// TIA Portal project "FactoryIO_Template_S7-1500_V15_parcial1_terminado1" (V15)

(* hardware
DEVICE "S71500/ET200MP-Station_1"  S7-1500 station
   slot 0: "Profilschiene_0"  6ES7 590-1***0-0AA0
   slot 1: "PLC_1"  CPU 1511-1 PN  6ES7 511-1AK00-0AB0  V1.8
   slot 2: "AI 8xU/I/RTD/TC ST_1"  AI 8xU/I/RTD/TC ST  6ES7 531-7KF00-0AB0  V2.0
   slot 3: "AI 8xU/I/RTD/TC ST_2"  AI 8xU/I/RTD/TC ST  6ES7 531-7KF00-0AB0  V2.0
   slot 4: "AI 8xU/I/RTD/TC ST_3"  AI 8xU/I/RTD/TC ST  6ES7 531-7KF00-0AB0  V2.0
   slot 5: "AI 8xU/I/RTD/TC ST_4"  AI 8xU/I/RTD/TC ST  6ES7 531-7KF00-0AB0  V2.0
   slot 6: "DI 16x24VDC BA_1"  DI 16x24VDC BA  6ES7 521-1BH10-0AA0  V1.0
*)

// ===== PLC "PLC_1"  CPU 1511-1 PN =====

VAR_GLOBAL   // PLC tag table "Standard-Variablentabelle"
   "Box_feeder" AT %Q0.0 : Bool;
   "Load_belt" AT %Q0.1 : Bool;
   "Start" AT %I0.0 : Bool;
   "Stop" AT %I0.1 : Bool;
   "Reset" AT %I0.2 : Bool;
   "Manual" AT %I0.3 : Bool;
   "Emergency_stop" AT %I0.5 : Bool;
   "Box_entry" AT %I0.6 : Bool;
   "Turn" AT %Q0.2 : Bool;
   "Pusher_limit" AT %I0.7 : Bool;
   "Push" AT %Q0.3 : Bool;
   "Open_Plate" AT %Q0.4 : Bool;
   "Plate_limit" AT %I1.0 : Bool;
   "Clamp" AT %Q0.5 : Bool;
   "Clamped" AT %I1.1 : Bool;
   "Pallet_feeder" AT %Q0.6 : Bool;
   "Pallet_at_entry" AT %I1.2 : Bool;
   "S1_Elevator_base" AT %I1.3 : Bool;
   "S2_Elevator_base" AT %I1.4 : Bool;
   "Pallet_at_exit" AT %I1.5 : Bool;
   "Exit_conveyor" AT %Q0.7 : Bool;
   "Elevator_moving" AT %I1.6 : Bool;
   "Move_to_limit" AT %Q1.0 : Bool;
   "Elevator_up" AT %Q1.1 : Bool;
   "Warning light" AT %Q1.3 : Bool;
   "Auto" AT %I0.4 : Bool;
   "Elevator_down" AT %Q1.2 : Bool;
   "Contador1" AT %MW10 : Int;
   "Contador2" AT %MW12 : Int;
   "Contador3" AT %MW14 : Int;
   "LimiteContador1" AT %MW20 : Int;
   "LimiteContador2" AT %MW22 : Int;
   "Pallet_in_acensor" AT %M100.0 : Bool;
   "Load_pallet" AT %Q1.4 : Bool;
   "Run_machine" AT %M0.0 : Bool;
   "Elevator_Listo_a_cargar" AT %M100.1 : Bool;
   "LimiteContador3" AT %MW24 : Int;
   "Plaforma_llena" AT %M100.2 : Bool;
   "Reposo" AT %M1000.0 : Bool;
   "Bandas_on" AT %M1000.1 : Bool;
   "Caja_en_posicion" AT %M1000.2 : Bool;
   "box_hacia_load_belt" AT %M1000.3 : Bool;
   "Avanzando_en_box_en_load_belt" AT %M1000.4 : Bool;
   "Haciendo_push" AT %M1000.5 : Bool;
   "Saliendo_push" AT %M1000.6 : Bool;
   "Push_afuera" AT %M1000.7 : Bool;
   "Push_regresando" AT %M1001.0 : Bool;
   "Push_en_inicio" AT %M1001.1 : Bool;
   "Cajas_en_plato" AT %M1001.2 : Bool;
   "Intercambiar_con_turn" AT %M1001.3 : Bool;
   "Intercambiar_sin_turn" AT %M1001.4 : Bool;
   "Reposo_inferiror" AT %M1100.0 : Bool;
   "Pallet_avanzando" AT %M1100.1 : Bool;
   "Entrando_a_load_pallet" AT %M1100.2 : Bool;
   "Pallet_en_posicion" AT %M1100.3 : Bool;
   "Acomodar_pallet" AT %M1100.4 : Bool;
   "Pallet_in_acesor_op" AT %M1100.5 : Bool;
   "Muevo_ascensor" AT %M1100.6 : Bool;
   "acesor_subiendo" AT %M1100.7 : Bool;
   "elevator_arriba" AT %M1101.0 : Bool;
   "Empezar_descarga_activar_clamp" AT %M1101.1 : Bool;
   "cajas_sujetas_a_descargar" AT %M1101.2 : Bool;
   "plate_abriendo" AT %M1101.3 : Bool;
   "plate_abierto" AT %M1101.4 : Bool;
   "Cajas_en_pallet" AT %M1101.5 : Bool;
   "elevator_bajando" AT %M1101.6 : Bool;
   "elevator_bajo_1" AT %M1101.7 : Bool;
   "Cerrando_plato" AT %M1102.0 : Bool;
   "plato_cerrado" AT %M1102.1 : Bool;
   "Elevador_lleno" AT %M1102.2 : Bool;
   "Acensor_bajando" AT %M1102.3 : Bool;
   "Asensor_abajo" AT %M1102.4 : Bool;
   "Pallet_Saliendo_de_elevador" AT %M1102.5 : Bool;
   "Restableciendo_inicio" AT %M1102.6 : Bool;
   "EstadosRdePCajas1" AT %MB1000 : Byte;
   "EstadosRdePEstibas1" AT %MB1100 : Byte;
   "EstadosRdePCajas2" AT %MB1001 : Byte;
   "MemEstadosRdePCajas1" AT %MB2000 : Byte;
   "MemEstadosRdePCajas2" AT %MB2001 : Byte;
   "MemEstadosRdePEstibas1" AT %MB2100 : Byte;
   "EstadosRdePEstibas2" AT %MB1101 : Byte;
   "EstadosRdePEstibas3" AT %MB1102 : Byte;
   "MemEstadosRdePEstibas2" AT %MB2101 : Byte;
   "MemEstadosRdePEstibas3" AT %MB2102 : Byte;
   "Salidas_Byte_0" AT %QB0 : Byte;
   "MemSalidas_Byte_0" AT %MB3000 : Byte;
   "Salidas_Byte_1" AT %QB1 : Byte;
   "MemSalidas_Byte_1" AT %MB3001 : Byte;
   "Tag_1" AT %M900.0 : Bool;
   "Tag_3" AT %M900.1 : Bool;
   "EstadosMaquina1" AT %MB100 : Byte;
   "MemEstadosMaquina1" AT %MB4000 : Byte;
   "Estado_On_Machine" AT %MB0 : Byte;
   "MenEstado_On_Machine" AT %MB5000 : Byte;
   "Entrada_POT" AT %ID30 : Real;
   "Salida_contador" AT %QD30 : Real;
   "Pot_int" AT %MW2 : Int;
   "Pallet_Feeder_Aux" AT %Q1.5 : Bool;
   "Roller_Stop" AT %Q1.6 : Bool;
END_VAR

// folder: System blocks/Program resources

DATA_BLOCK "Contador_1"   // DB1
{ S7_Optimized_Access := 'TRUE' }
AUTHOR : Simatic
FAMILY : IEC
NAME : CNTR
VERSION : 1.0
// stored: InstanceOfName IEC_COUNTER
"IEC_COUNTER"
BEGIN
END_DATA_BLOCK

DATA_BLOCK "Contador_2"   // DB2
{ S7_Optimized_Access := 'TRUE' }
AUTHOR : Simatic
FAMILY : IEC
NAME : CNTR
VERSION : 1.0
// stored: InstanceOfName IEC_COUNTER
"IEC_COUNTER"
BEGIN
END_DATA_BLOCK

DATA_BLOCK "Contador_3"   // DB3
{ S7_Optimized_Access := 'TRUE' }
AUTHOR : Simatic
FAMILY : IEC
NAME : CNTR
VERSION : 1.0
// stored: InstanceOfName IEC_COUNTER
"IEC_COUNTER"
BEGIN
END_DATA_BLOCK

// folder: (top level)

FUNCTION "Nivel_superior" : Void   // FC1, LAD
{ S7_Optimized_Access := 'TRUE' }
VERSION : 0.1
   VAR_TEMP   // added for the SCL form of the ladder/FBD networks
      _w1 : Bool;
   END_VAR
BEGIN

REGION Network 1
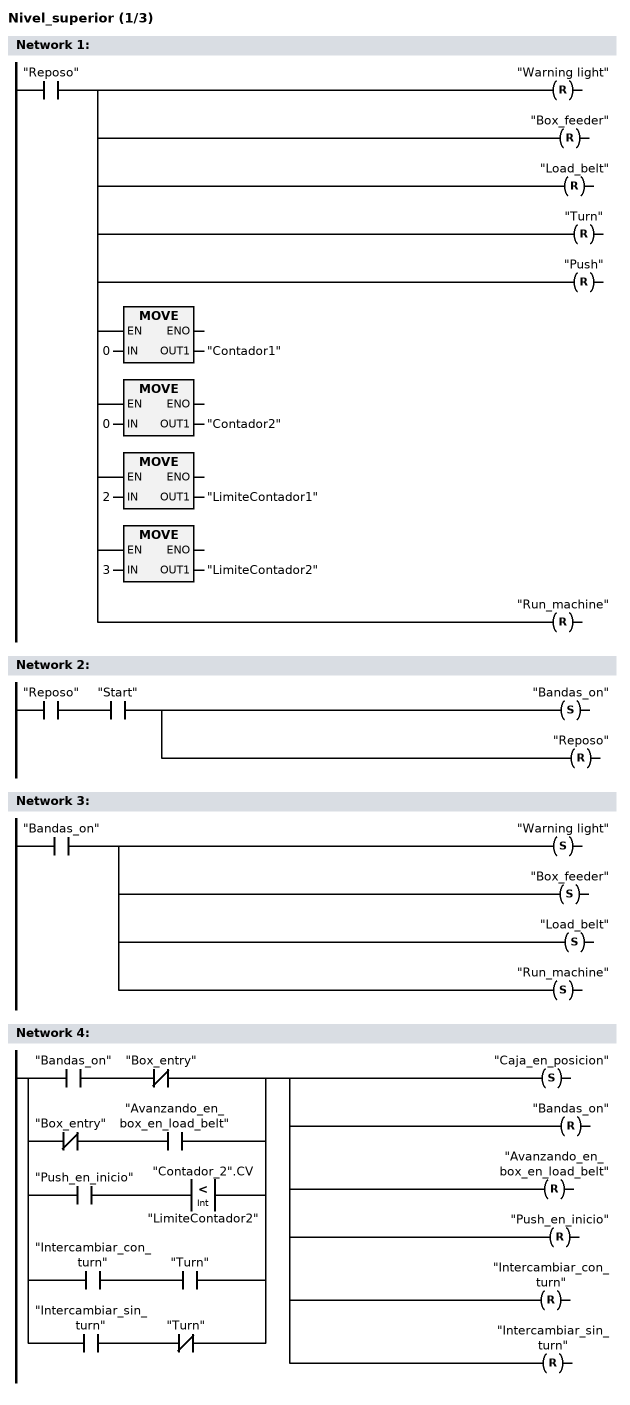
   RUNG wire#powerrail
      Contact( "Reposo" )
      wire#w1
      R_Coil( "Warning light" )
   END_RUNG
   RUNG wire#w1
      R_Coil( "Box_feeder" )
   END_RUNG
   RUNG wire#w1
      R_Coil( "Load_belt" )
   END_RUNG
   RUNG wire#w1
      R_Coil( "Turn" )
   END_RUNG
   RUNG wire#w1
      R_Coil( "Push" )
   END_RUNG
   RUNG wire#w1
      Move(in := 0, out1 => "Contador1")
   END_RUNG
   RUNG wire#w1
      Move(in := 0, out1 => "Contador2")
   END_RUNG
   RUNG wire#w1
      Move(in := 2, out1 => "LimiteContador1")
   END_RUNG
   RUNG wire#w1
      Move(in := 3, out1 => "LimiteContador2")
   END_RUNG
   RUNG wire#w1
      R_Coil( "Run_machine" )
   END_RUNG
   // the same network as SCL:
   IF "Reposo" THEN
       "Warning light" := FALSE;
       "Box_feeder" := FALSE;
       "Load_belt" := FALSE;
       "Turn" := FALSE;
       "Push" := FALSE;
       "Contador1" := 0;
       "Contador2" := 0;
       "LimiteContador1" := 2;
       "LimiteContador2" := 3;
       "Run_machine" := FALSE;
   END_IF;
END_REGION

REGION Network 2
   RUNG wire#powerrail
      Contact( "Reposo" )
      Contact( "Start" )
      wire#w1
      S_Coil( "Bandas_on" )
   END_RUNG
   RUNG wire#w1
      R_Coil( "Reposo" )
   END_RUNG
   // the same network as SCL:
   IF "Reposo" AND "Start" THEN
       "Bandas_on" := TRUE;
       "Reposo" := FALSE;
   END_IF;
END_REGION

REGION Network 3
   RUNG wire#powerrail
      Contact( "Bandas_on" )
      wire#w1
      S_Coil( "Warning light" )
   END_RUNG
   RUNG wire#w1
      S_Coil( "Box_feeder" )
   END_RUNG
   RUNG wire#w1
      S_Coil( "Load_belt" )
   END_RUNG
   RUNG wire#w1
      S_Coil( "Run_machine" )
   END_RUNG
   // the same network as SCL:
   IF "Bandas_on" THEN
       "Warning light" := TRUE;
       "Box_feeder" := TRUE;
       "Load_belt" := TRUE;
       "Run_machine" := TRUE;
   END_IF;
END_REGION

REGION Network 4
   RUNG wire#powerrail
      Contact( "Bandas_on" )
      I_Contact( "Box_entry" )
      wire#w1
      S_Coil( "Caja_en_posicion" )
   END_RUNG
   RUNG wire#powerrail
      I_Contact( "Box_entry" )
      Contact( "Avanzando_en_box_en_load_belt" )
   END_RUNG wire#w1
   RUNG wire#powerrail
      Contact( "Push_en_inicio" )
      { S7_Templates := "SrcType := Int" } LT_Contact(in1 := "Contador_2".CV, in2 := "LimiteContador2")
   END_RUNG wire#w1
   RUNG wire#powerrail
      Contact( "Intercambiar_con_turn" )
      Contact( "Turn" )
   END_RUNG wire#w1
   RUNG wire#powerrail
      Contact( "Intercambiar_sin_turn" )
      I_Contact( "Turn" )
   END_RUNG wire#w1
   RUNG wire#w1
      R_Coil( "Bandas_on" )
   END_RUNG
   RUNG wire#w1
      R_Coil( "Avanzando_en_box_en_load_belt" )
   END_RUNG
   RUNG wire#w1
      R_Coil( "Push_en_inicio" )
   END_RUNG
   RUNG wire#w1
      R_Coil( "Intercambiar_con_turn" )
   END_RUNG
   RUNG wire#w1
      R_Coil( "Intercambiar_sin_turn" )
   END_RUNG
   // the same network as SCL:
   IF ("Bandas_on" AND NOT "Box_entry") OR (NOT "Box_entry" AND "Avanzando_en_box_en_load_belt") OR ("Push_en_inicio" AND ("Contador_2".CV < "LimiteContador2")) OR ("Intercambiar_con_turn" AND "Turn") OR ("Intercambiar_sin_turn" AND NOT "Turn") THEN
       "Caja_en_posicion" := TRUE;
   END_IF;
   #_w1 := ("Bandas_on" AND NOT "Box_entry") OR (NOT "Box_entry" AND "Avanzando_en_box_en_load_belt") OR ("Push_en_inicio" AND ("Contador_2".CV < "LimiteContador2")) OR ("Intercambiar_con_turn" AND "Turn") OR ("Intercambiar_sin_turn" AND NOT "Turn");
   IF #_w1 THEN
       "Bandas_on" := FALSE;
       "Avanzando_en_box_en_load_belt" := FALSE;
       "Push_en_inicio" := FALSE;
       "Intercambiar_con_turn" := FALSE;
       "Intercambiar_sin_turn" := FALSE;
   END_IF;
END_REGION

REGION Network 5
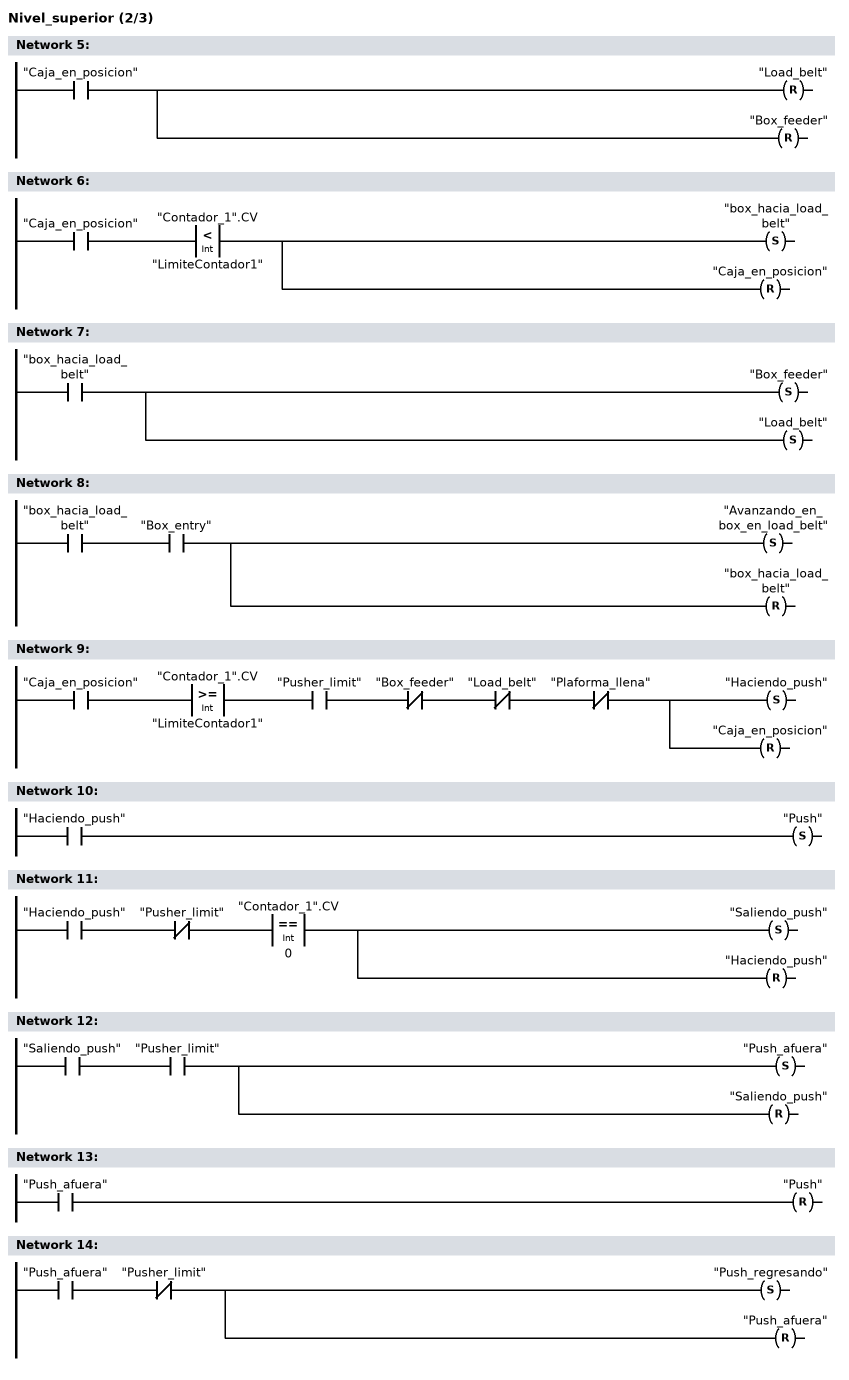
   RUNG wire#powerrail
      Contact( "Caja_en_posicion" )
      wire#w1
      R_Coil( "Load_belt" )
   END_RUNG
   RUNG wire#w1
      R_Coil( "Box_feeder" )
   END_RUNG
   // the same network as SCL:
   IF "Caja_en_posicion" THEN
       "Load_belt" := FALSE;
       "Box_feeder" := FALSE;
   END_IF;
END_REGION

REGION Network 6
   RUNG wire#powerrail
      Contact( "Caja_en_posicion" )
      { S7_Templates := "SrcType := Int" } LT_Contact(in1 := "Contador_1".CV, in2 := "LimiteContador1")
      wire#w1
      S_Coil( "box_hacia_load_belt" )
   END_RUNG
   RUNG wire#w1
      R_Coil( "Caja_en_posicion" )
   END_RUNG
   // the same network as SCL:
   IF "Caja_en_posicion" AND ("Contador_1".CV < "LimiteContador1") THEN
       "box_hacia_load_belt" := TRUE;
       "Caja_en_posicion" := FALSE;
   END_IF;
END_REGION

REGION Network 7
   RUNG wire#powerrail
      Contact( "box_hacia_load_belt" )
      wire#w1
      S_Coil( "Box_feeder" )
   END_RUNG
   RUNG wire#w1
      S_Coil( "Load_belt" )
   END_RUNG
   // the same network as SCL:
   IF "box_hacia_load_belt" THEN
       "Box_feeder" := TRUE;
       "Load_belt" := TRUE;
   END_IF;
END_REGION

REGION Network 8
   RUNG wire#powerrail
      Contact( "box_hacia_load_belt" )
      Contact( "Box_entry" )
      wire#w1
      S_Coil( "Avanzando_en_box_en_load_belt" )
   END_RUNG
   RUNG wire#w1
      R_Coil( "box_hacia_load_belt" )
   END_RUNG
   // the same network as SCL:
   IF "box_hacia_load_belt" AND "Box_entry" THEN
       "Avanzando_en_box_en_load_belt" := TRUE;
       "box_hacia_load_belt" := FALSE;
   END_IF;
END_REGION

REGION Network 9
   RUNG wire#powerrail
      Contact( "Caja_en_posicion" )
      { S7_Templates := "SrcType := Int" } GE_Contact(in1 := "Contador_1".CV, in2 := "LimiteContador1")
      Contact( "Pusher_limit" )
      I_Contact( "Box_feeder" )
      I_Contact( "Load_belt" )
      I_Contact( "Plaforma_llena" )
      wire#w1
      S_Coil( "Haciendo_push" )
   END_RUNG
   RUNG wire#w1
      R_Coil( "Caja_en_posicion" )
   END_RUNG
   // the same network as SCL:
   IF "Caja_en_posicion" AND ("Contador_1".CV >= "LimiteContador1") AND "Pusher_limit" AND NOT "Box_feeder" AND NOT "Load_belt" AND NOT "Plaforma_llena" THEN
       "Haciendo_push" := TRUE;
       "Caja_en_posicion" := FALSE;
   END_IF;
END_REGION

REGION Network 10
   RUNG wire#powerrail
      Contact( "Haciendo_push" )
      S_Coil( "Push" )
   END_RUNG
   // the same network as SCL:
   IF "Haciendo_push" THEN "Push" := TRUE; END_IF;
END_REGION

REGION Network 11
   RUNG wire#powerrail
      Contact( "Haciendo_push" )
      I_Contact( "Pusher_limit" )
      { S7_Templates := "SrcType := Int" } EQ_Contact(in1 := "Contador_1".CV, in2 := 0)
      wire#w1
      S_Coil( "Saliendo_push" )
   END_RUNG
   RUNG wire#w1
      R_Coil( "Haciendo_push" )
   END_RUNG
   // the same network as SCL:
   IF "Haciendo_push" AND NOT "Pusher_limit" AND ("Contador_1".CV = 0) THEN
       "Saliendo_push" := TRUE;
       "Haciendo_push" := FALSE;
   END_IF;
END_REGION

REGION Network 12
   RUNG wire#powerrail
      Contact( "Saliendo_push" )
      Contact( "Pusher_limit" )
      wire#w1
      S_Coil( "Push_afuera" )
   END_RUNG
   RUNG wire#w1
      R_Coil( "Saliendo_push" )
   END_RUNG
   // the same network as SCL:
   IF "Saliendo_push" AND "Pusher_limit" THEN
       "Push_afuera" := TRUE;
       "Saliendo_push" := FALSE;
   END_IF;
END_REGION

REGION Network 13
   RUNG wire#powerrail
      Contact( "Push_afuera" )
      R_Coil( "Push" )
   END_RUNG
   // the same network as SCL:
   IF "Push_afuera" THEN "Push" := FALSE; END_IF;
END_REGION

REGION Network 14
   RUNG wire#powerrail
      Contact( "Push_afuera" )
      I_Contact( "Pusher_limit" )
      wire#w1
      S_Coil( "Push_regresando" )
   END_RUNG
   RUNG wire#w1
      R_Coil( "Push_afuera" )
   END_RUNG
   // the same network as SCL:
   IF "Push_afuera" AND NOT "Pusher_limit" THEN
       "Push_regresando" := TRUE;
       "Push_afuera" := FALSE;
   END_IF;
END_REGION

REGION Network 15
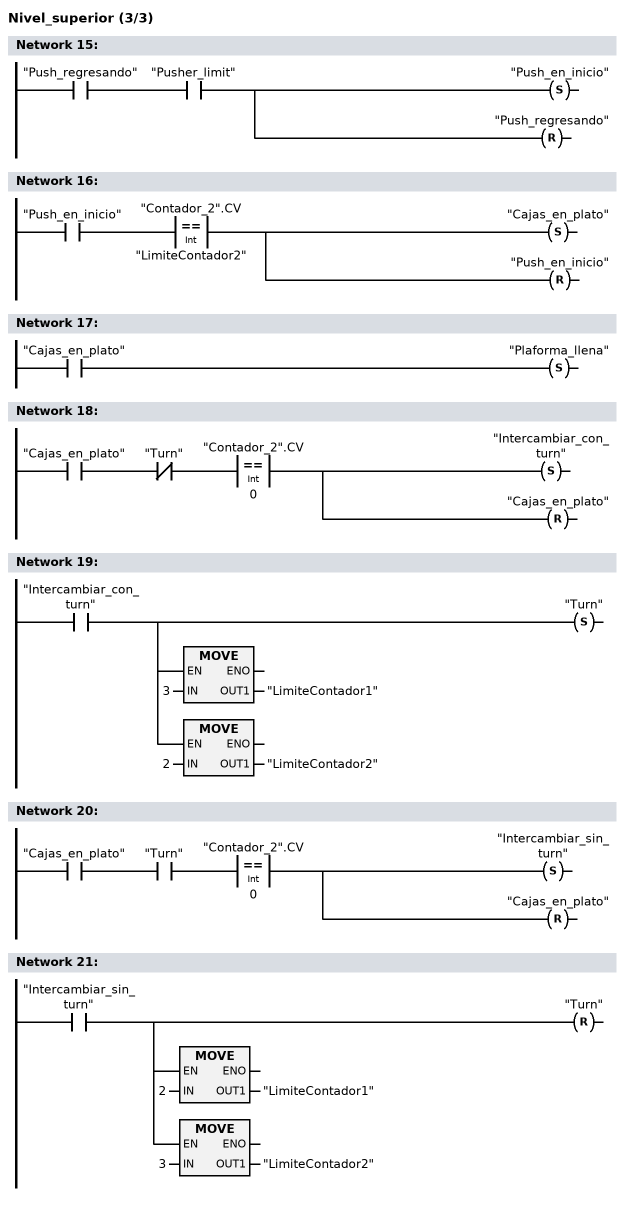
   RUNG wire#powerrail
      Contact( "Push_regresando" )
      Contact( "Pusher_limit" )
      wire#w1
      S_Coil( "Push_en_inicio" )
   END_RUNG
   RUNG wire#w1
      R_Coil( "Push_regresando" )
   END_RUNG
   // the same network as SCL:
   IF "Push_regresando" AND "Pusher_limit" THEN
       "Push_en_inicio" := TRUE;
       "Push_regresando" := FALSE;
   END_IF;
END_REGION

REGION Network 16
   RUNG wire#powerrail
      Contact( "Push_en_inicio" )
      { S7_Templates := "SrcType := Int" } EQ_Contact(in1 := "Contador_2".CV, in2 := "LimiteContador2")
      wire#w1
      S_Coil( "Cajas_en_plato" )
   END_RUNG
   RUNG wire#w1
      R_Coil( "Push_en_inicio" )
   END_RUNG
   // the same network as SCL:
   IF "Push_en_inicio" AND ("Contador_2".CV = "LimiteContador2") THEN
       "Cajas_en_plato" := TRUE;
       "Push_en_inicio" := FALSE;
   END_IF;
END_REGION

REGION Network 17
   RUNG wire#powerrail
      Contact( "Cajas_en_plato" )
      S_Coil( "Plaforma_llena" )
   END_RUNG
   // the same network as SCL:
   IF "Cajas_en_plato" THEN "Plaforma_llena" := TRUE; END_IF;
END_REGION

REGION Network 18
   RUNG wire#powerrail
      Contact( "Cajas_en_plato" )
      I_Contact( "Turn" )
      { S7_Templates := "SrcType := Int" } EQ_Contact(in1 := "Contador_2".CV, in2 := 0)
      wire#w1
      S_Coil( "Intercambiar_con_turn" )
   END_RUNG
   RUNG wire#w1
      R_Coil( "Cajas_en_plato" )
   END_RUNG
   // the same network as SCL:
   IF "Cajas_en_plato" AND NOT "Turn" AND ("Contador_2".CV = 0) THEN
       "Intercambiar_con_turn" := TRUE;
       "Cajas_en_plato" := FALSE;
   END_IF;
END_REGION

REGION Network 19
   RUNG wire#powerrail
      Contact( "Intercambiar_con_turn" )
      wire#w1
      S_Coil( "Turn" )
   END_RUNG
   RUNG wire#w1
      Move(in := 3, out1 => "LimiteContador1")
   END_RUNG
   RUNG wire#w1
      Move(in := 2, out1 => "LimiteContador2")
   END_RUNG
   // the same network as SCL:
   IF "Intercambiar_con_turn" THEN
       "Turn" := TRUE;
       "LimiteContador1" := 3;
       "LimiteContador2" := 2;
   END_IF;
END_REGION

REGION Network 20
   RUNG wire#powerrail
      Contact( "Cajas_en_plato" )
      Contact( "Turn" )
      { S7_Templates := "SrcType := Int" } EQ_Contact(in1 := "Contador_2".CV, in2 := 0)
      wire#w1
      S_Coil( "Intercambiar_sin_turn" )
   END_RUNG
   RUNG wire#w1
      R_Coil( "Cajas_en_plato" )
   END_RUNG
   // the same network as SCL:
   IF "Cajas_en_plato" AND "Turn" AND ("Contador_2".CV = 0) THEN
       "Intercambiar_sin_turn" := TRUE;
       "Cajas_en_plato" := FALSE;
   END_IF;
END_REGION

REGION Network 21
   RUNG wire#powerrail
      Contact( "Intercambiar_sin_turn" )
      wire#w1
      R_Coil( "Turn" )
   END_RUNG
   RUNG wire#w1
      Move(in := 2, out1 => "LimiteContador1")
   END_RUNG
   RUNG wire#w1
      Move(in := 3, out1 => "LimiteContador2")
   END_RUNG
   // the same network as SCL:
   IF "Intercambiar_sin_turn" THEN
       "Turn" := FALSE;
       "LimiteContador1" := 2;
       "LimiteContador2" := 3;
   END_IF;
END_REGION
END_FUNCTION

FUNCTION "Nivel_inferior" : Void   // FC2, LAD
{ S7_Optimized_Access := 'TRUE' }
VERSION : 0.1
   VAR_TEMP   // added for the SCL form of the ladder/FBD networks
      _w1 : Bool;
   END_VAR
BEGIN

REGION Network 1
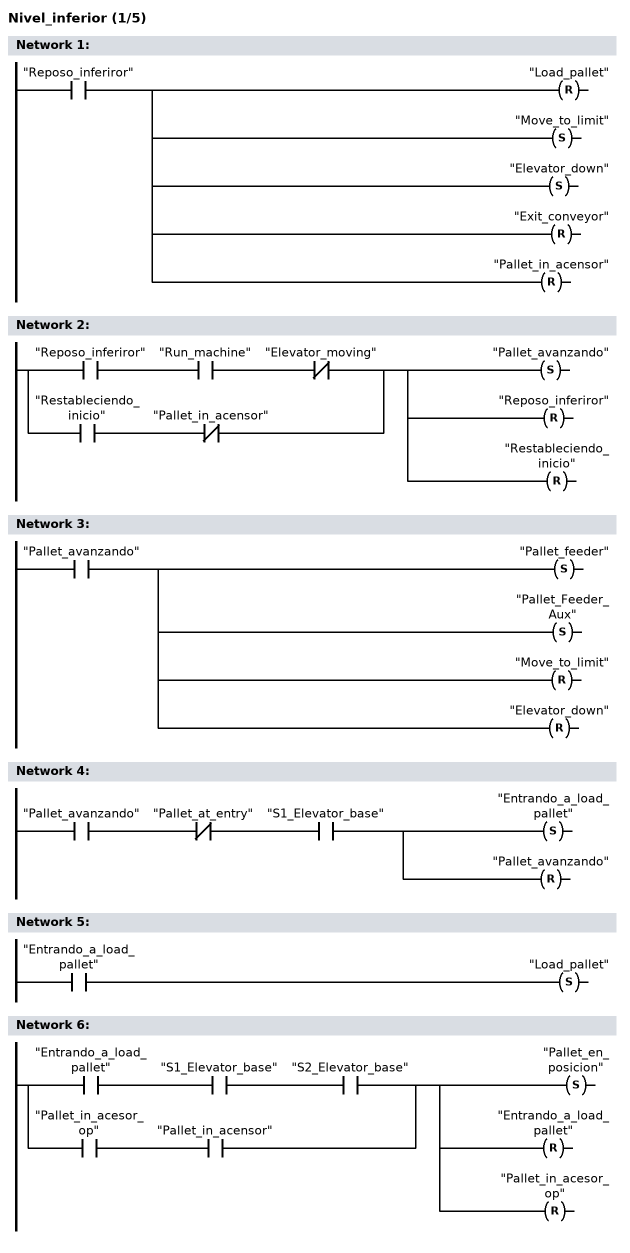
   RUNG wire#powerrail
      Contact( "Reposo_inferiror" )
      wire#w1
      R_Coil( "Load_pallet" )
   END_RUNG
   RUNG wire#w1
      S_Coil( "Move_to_limit" )
   END_RUNG
   RUNG wire#w1
      S_Coil( "Elevator_down" )
   END_RUNG
   RUNG wire#w1
      R_Coil( "Exit_conveyor" )
   END_RUNG
   RUNG wire#w1
      R_Coil( "Pallet_in_acensor" )
   END_RUNG
   // the same network as SCL:
   IF "Reposo_inferiror" THEN
       "Load_pallet" := FALSE;
       "Move_to_limit" := TRUE;
       "Elevator_down" := TRUE;
       "Exit_conveyor" := FALSE;
       "Pallet_in_acensor" := FALSE;
   END_IF;
END_REGION

REGION Network 2
   RUNG wire#powerrail
      Contact( "Reposo_inferiror" )
      Contact( "Run_machine" )
      I_Contact( "Elevator_moving" )
      wire#w1
      S_Coil( "Pallet_avanzando" )
   END_RUNG
   RUNG wire#powerrail
      Contact( "Restableciendo_inicio" )
      I_Contact( "Pallet_in_acensor" )
   END_RUNG wire#w1
   RUNG wire#w1
      R_Coil( "Reposo_inferiror" )
   END_RUNG
   RUNG wire#w1
      R_Coil( "Restableciendo_inicio" )
   END_RUNG
   // the same network as SCL:
   IF ("Reposo_inferiror" AND "Run_machine" AND NOT "Elevator_moving") OR ("Restableciendo_inicio" AND NOT "Pallet_in_acensor") THEN
       "Pallet_avanzando" := TRUE;
   END_IF;
   #_w1 := ("Reposo_inferiror" AND "Run_machine" AND NOT "Elevator_moving") OR ("Restableciendo_inicio" AND NOT "Pallet_in_acensor");
   IF #_w1 THEN
       "Reposo_inferiror" := FALSE;
       "Restableciendo_inicio" := FALSE;
   END_IF;
END_REGION

REGION Network 3
   RUNG wire#powerrail
      Contact( "Pallet_avanzando" )
      wire#w1
      S_Coil( "Pallet_feeder" )
   END_RUNG
   RUNG wire#w1
      S_Coil( "Pallet_Feeder_Aux" )
   END_RUNG
   RUNG wire#w1
      R_Coil( "Move_to_limit" )
   END_RUNG
   RUNG wire#w1
      R_Coil( "Elevator_down" )
   END_RUNG
   // the same network as SCL:
   IF "Pallet_avanzando" THEN
       "Pallet_feeder" := TRUE;
       "Pallet_Feeder_Aux" := TRUE;
       "Move_to_limit" := FALSE;
       "Elevator_down" := FALSE;
   END_IF;
END_REGION

REGION Network 4
   RUNG wire#powerrail
      Contact( "Pallet_avanzando" )
      I_Contact( "Pallet_at_entry" )
      Contact( "S1_Elevator_base" )
      wire#w1
      S_Coil( "Entrando_a_load_pallet" )
   END_RUNG
   RUNG wire#w1
      R_Coil( "Pallet_avanzando" )
   END_RUNG
   // the same network as SCL:
   IF "Pallet_avanzando" AND NOT "Pallet_at_entry" AND "S1_Elevator_base" THEN
       "Entrando_a_load_pallet" := TRUE;
       "Pallet_avanzando" := FALSE;
   END_IF;
END_REGION

REGION Network 5
   RUNG wire#powerrail
      Contact( "Entrando_a_load_pallet" )
      S_Coil( "Load_pallet" )
   END_RUNG
   // the same network as SCL:
   IF "Entrando_a_load_pallet" THEN "Load_pallet" := TRUE; END_IF;
END_REGION

REGION Network 6
   RUNG wire#powerrail
      Contact( "Entrando_a_load_pallet" )
      Contact( "S1_Elevator_base" )
      Contact( "S2_Elevator_base" )
      wire#w1
      S_Coil( "Pallet_en_posicion" )
   END_RUNG
   RUNG wire#powerrail
      Contact( "Pallet_in_acesor_op" )
      Contact( "Pallet_in_acensor" )
   END_RUNG wire#w1
   RUNG wire#w1
      R_Coil( "Entrando_a_load_pallet" )
   END_RUNG
   RUNG wire#w1
      R_Coil( "Pallet_in_acesor_op" )
   END_RUNG
   // the same network as SCL:
   IF ("Entrando_a_load_pallet" AND "S1_Elevator_base" AND "S2_Elevator_base") OR ("Pallet_in_acesor_op" AND "Pallet_in_acensor") THEN
       "Pallet_en_posicion" := TRUE;
   END_IF;
   #_w1 := ("Entrando_a_load_pallet" AND "S1_Elevator_base" AND "S2_Elevator_base") OR ("Pallet_in_acesor_op" AND "Pallet_in_acensor");
   IF #_w1 THEN
       "Entrando_a_load_pallet" := FALSE;
       "Pallet_in_acesor_op" := FALSE;
   END_IF;
END_REGION

REGION Network 7
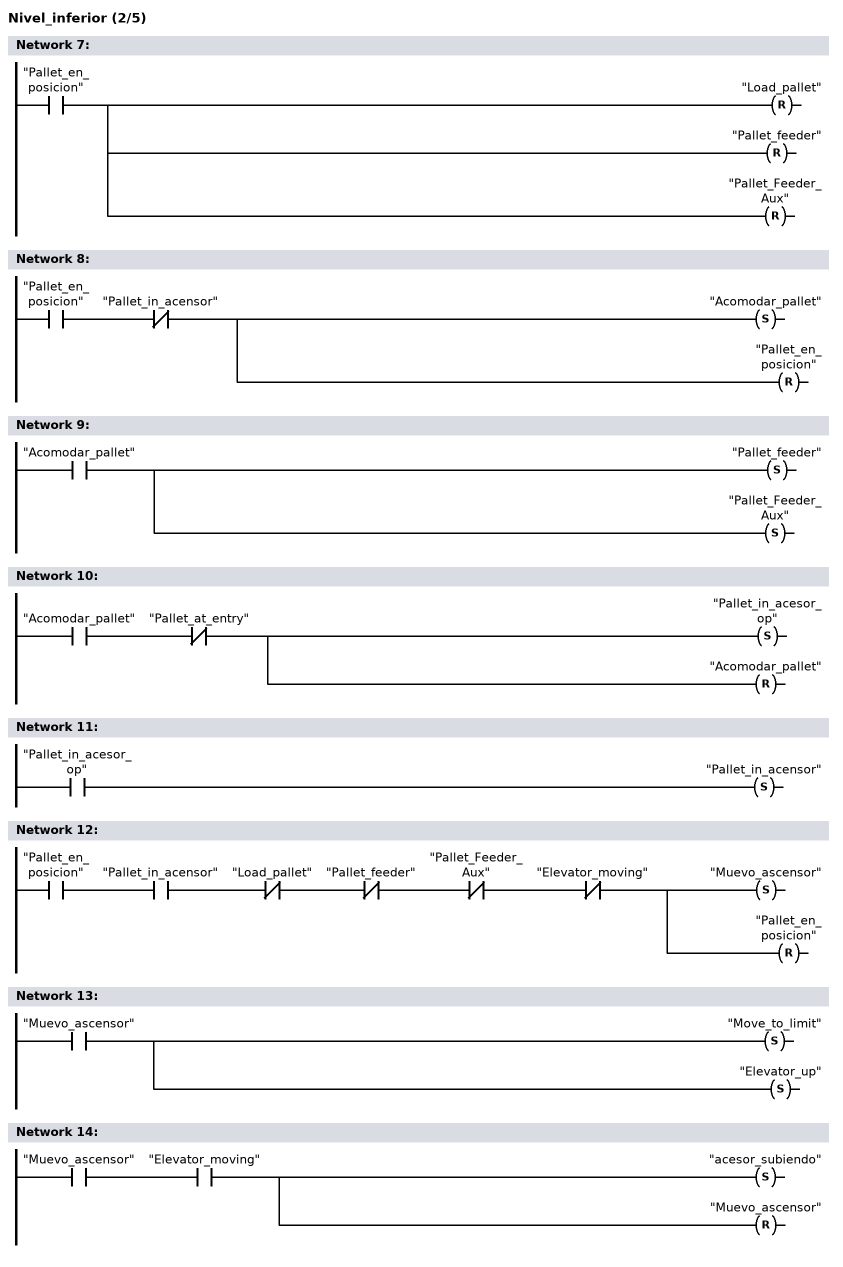
   RUNG wire#powerrail
      Contact( "Pallet_en_posicion" )
      wire#w1
      R_Coil( "Load_pallet" )
   END_RUNG
   RUNG wire#w1
      R_Coil( "Pallet_feeder" )
   END_RUNG
   RUNG wire#w1
      R_Coil( "Pallet_Feeder_Aux" )
   END_RUNG
   // the same network as SCL:
   IF "Pallet_en_posicion" THEN
       "Load_pallet" := FALSE;
       "Pallet_feeder" := FALSE;
       "Pallet_Feeder_Aux" := FALSE;
   END_IF;
END_REGION

REGION Network 8
   RUNG wire#powerrail
      Contact( "Pallet_en_posicion" )
      I_Contact( "Pallet_in_acensor" )
      wire#w1
      S_Coil( "Acomodar_pallet" )
   END_RUNG
   RUNG wire#w1
      R_Coil( "Pallet_en_posicion" )
   END_RUNG
   // the same network as SCL:
   IF "Pallet_en_posicion" AND NOT "Pallet_in_acensor" THEN
       "Acomodar_pallet" := TRUE;
       "Pallet_en_posicion" := FALSE;
   END_IF;
END_REGION

REGION Network 9
   RUNG wire#powerrail
      Contact( "Acomodar_pallet" )
      wire#w1
      S_Coil( "Pallet_feeder" )
   END_RUNG
   RUNG wire#w1
      S_Coil( "Pallet_Feeder_Aux" )
   END_RUNG
   // the same network as SCL:
   IF "Acomodar_pallet" THEN
       "Pallet_feeder" := TRUE;
       "Pallet_Feeder_Aux" := TRUE;
   END_IF;
END_REGION

REGION Network 10
   RUNG wire#powerrail
      Contact( "Acomodar_pallet" )
      I_Contact( "Pallet_at_entry" )
      wire#w1
      S_Coil( "Pallet_in_acesor_op" )
   END_RUNG
   RUNG wire#w1
      R_Coil( "Acomodar_pallet" )
   END_RUNG
   // the same network as SCL:
   IF "Acomodar_pallet" AND NOT "Pallet_at_entry" THEN
       "Pallet_in_acesor_op" := TRUE;
       "Acomodar_pallet" := FALSE;
   END_IF;
END_REGION

REGION Network 11
   RUNG wire#powerrail
      Contact( "Pallet_in_acesor_op" )
      S_Coil( "Pallet_in_acensor" )
   END_RUNG
   // the same network as SCL:
   IF "Pallet_in_acesor_op" THEN "Pallet_in_acensor" := TRUE; END_IF;
END_REGION

REGION Network 12
   RUNG wire#powerrail
      Contact( "Pallet_en_posicion" )
      Contact( "Pallet_in_acensor" )
      I_Contact( "Load_pallet" )
      I_Contact( "Pallet_feeder" )
      I_Contact( "Pallet_Feeder_Aux" )
      I_Contact( "Elevator_moving" )
      wire#w1
      S_Coil( "Muevo_ascensor" )
   END_RUNG
   RUNG wire#w1
      R_Coil( "Pallet_en_posicion" )
   END_RUNG
   // the same network as SCL:
   IF "Pallet_en_posicion" AND "Pallet_in_acensor" AND NOT "Load_pallet" AND NOT "Pallet_feeder" AND NOT "Pallet_Feeder_Aux" AND NOT "Elevator_moving" THEN
       "Muevo_ascensor" := TRUE;
       "Pallet_en_posicion" := FALSE;
   END_IF;
END_REGION

REGION Network 13
   RUNG wire#powerrail
      Contact( "Muevo_ascensor" )
      wire#w1
      S_Coil( "Move_to_limit" )
   END_RUNG
   RUNG wire#w1
      S_Coil( "Elevator_up" )
   END_RUNG
   // the same network as SCL:
   IF "Muevo_ascensor" THEN
       "Move_to_limit" := TRUE;
       "Elevator_up" := TRUE;
   END_IF;
END_REGION

REGION Network 14
   RUNG wire#powerrail
      Contact( "Muevo_ascensor" )
      Contact( "Elevator_moving" )
      wire#w1
      S_Coil( "acesor_subiendo" )
   END_RUNG
   RUNG wire#w1
      R_Coil( "Muevo_ascensor" )
   END_RUNG
   // the same network as SCL:
   IF "Muevo_ascensor" AND "Elevator_moving" THEN
       "acesor_subiendo" := TRUE;
       "Muevo_ascensor" := FALSE;
   END_IF;
END_REGION

REGION Network 15
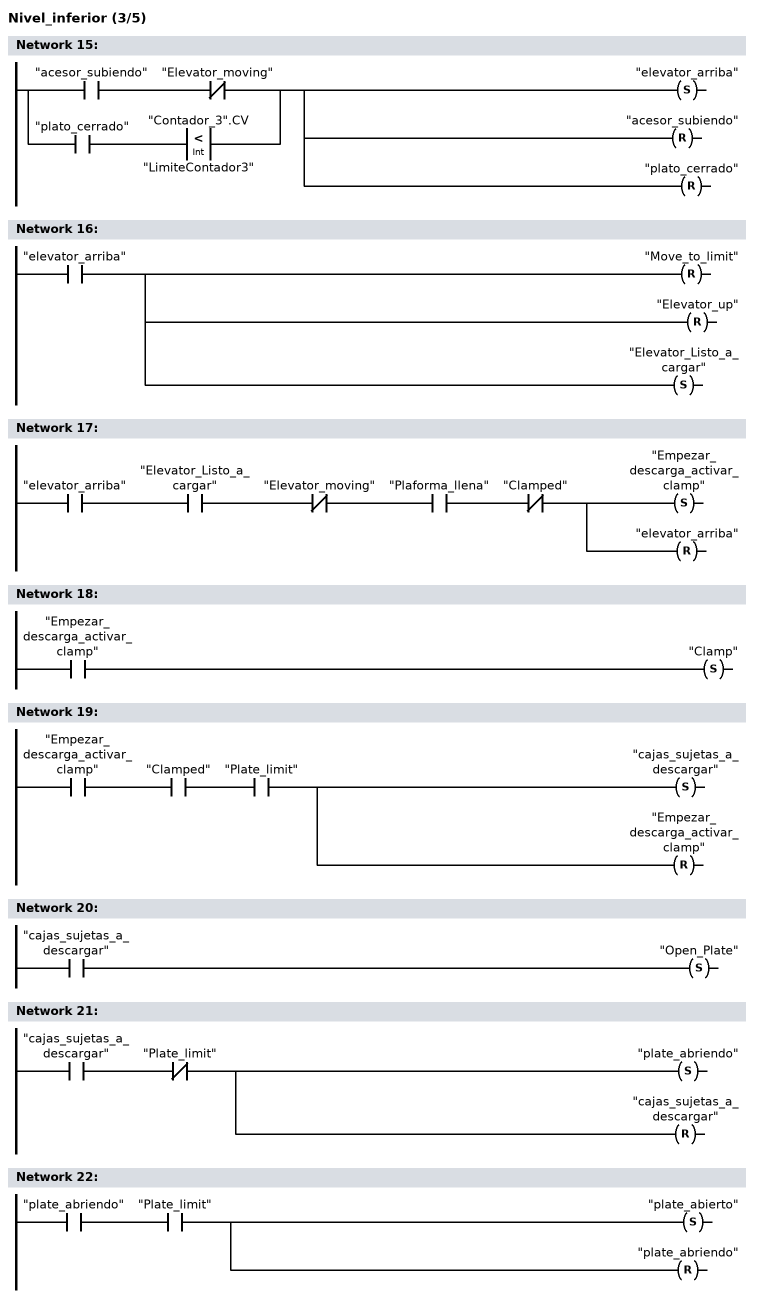
   RUNG wire#powerrail
      Contact( "acesor_subiendo" )
      I_Contact( "Elevator_moving" )
      wire#w1
      S_Coil( "elevator_arriba" )
   END_RUNG
   RUNG wire#powerrail
      Contact( "plato_cerrado" )
      { S7_Templates := "SrcType := Int" } LT_Contact(in1 := "Contador_3".CV, in2 := "LimiteContador3")
   END_RUNG wire#w1
   RUNG wire#w1
      R_Coil( "acesor_subiendo" )
   END_RUNG
   RUNG wire#w1
      R_Coil( "plato_cerrado" )
   END_RUNG
   // the same network as SCL:
   IF ("acesor_subiendo" AND NOT "Elevator_moving") OR ("plato_cerrado" AND ("Contador_3".CV < "LimiteContador3")) THEN
       "elevator_arriba" := TRUE;
   END_IF;
   #_w1 := ("acesor_subiendo" AND NOT "Elevator_moving") OR ("plato_cerrado" AND ("Contador_3".CV < "LimiteContador3"));
   IF #_w1 THEN
       "acesor_subiendo" := FALSE;
       "plato_cerrado" := FALSE;
   END_IF;
END_REGION

REGION Network 16
   RUNG wire#powerrail
      Contact( "elevator_arriba" )
      wire#w1
      R_Coil( "Move_to_limit" )
   END_RUNG
   RUNG wire#w1
      R_Coil( "Elevator_up" )
   END_RUNG
   RUNG wire#w1
      S_Coil( "Elevator_Listo_a_cargar" )
   END_RUNG
   // the same network as SCL:
   IF "elevator_arriba" THEN
       "Move_to_limit" := FALSE;
       "Elevator_up" := FALSE;
       "Elevator_Listo_a_cargar" := TRUE;
   END_IF;
END_REGION

REGION Network 17
   RUNG wire#powerrail
      Contact( "elevator_arriba" )
      Contact( "Elevator_Listo_a_cargar" )
      I_Contact( "Elevator_moving" )
      Contact( "Plaforma_llena" )
      I_Contact( "Clamped" )
      wire#w1
      S_Coil( "Empezar_descarga_activar_clamp" )
   END_RUNG
   RUNG wire#w1
      R_Coil( "elevator_arriba" )
   END_RUNG
   // the same network as SCL:
   IF "elevator_arriba" AND "Elevator_Listo_a_cargar" AND NOT "Elevator_moving" AND "Plaforma_llena" AND NOT "Clamped" THEN
       "Empezar_descarga_activar_clamp" := TRUE;
       "elevator_arriba" := FALSE;
   END_IF;
END_REGION

REGION Network 18
   RUNG wire#powerrail
      Contact( "Empezar_descarga_activar_clamp" )
      S_Coil( "Clamp" )
   END_RUNG
   // the same network as SCL:
   IF "Empezar_descarga_activar_clamp" THEN "Clamp" := TRUE; END_IF;
END_REGION

REGION Network 19
   RUNG wire#powerrail
      Contact( "Empezar_descarga_activar_clamp" )
      Contact( "Clamped" )
      Contact( "Plate_limit" )
      wire#w1
      S_Coil( "cajas_sujetas_a_descargar" )
   END_RUNG
   RUNG wire#w1
      R_Coil( "Empezar_descarga_activar_clamp" )
   END_RUNG
   // the same network as SCL:
   IF "Empezar_descarga_activar_clamp" AND "Clamped" AND "Plate_limit" THEN
       "cajas_sujetas_a_descargar" := TRUE;
       "Empezar_descarga_activar_clamp" := FALSE;
   END_IF;
END_REGION

REGION Network 20
   RUNG wire#powerrail
      Contact( "cajas_sujetas_a_descargar" )
      S_Coil( "Open_Plate" )
   END_RUNG
   // the same network as SCL:
   IF "cajas_sujetas_a_descargar" THEN "Open_Plate" := TRUE; END_IF;
END_REGION

REGION Network 21
   RUNG wire#powerrail
      Contact( "cajas_sujetas_a_descargar" )
      I_Contact( "Plate_limit" )
      wire#w1
      S_Coil( "plate_abriendo" )
   END_RUNG
   RUNG wire#w1
      R_Coil( "cajas_sujetas_a_descargar" )
   END_RUNG
   // the same network as SCL:
   IF "cajas_sujetas_a_descargar" AND NOT "Plate_limit" THEN
       "plate_abriendo" := TRUE;
       "cajas_sujetas_a_descargar" := FALSE;
   END_IF;
END_REGION

REGION Network 22
   RUNG wire#powerrail
      Contact( "plate_abriendo" )
      Contact( "Plate_limit" )
      wire#w1
      S_Coil( "plate_abierto" )
   END_RUNG
   RUNG wire#w1
      R_Coil( "plate_abriendo" )
   END_RUNG
   // the same network as SCL:
   IF "plate_abriendo" AND "Plate_limit" THEN
       "plate_abierto" := TRUE;
       "plate_abriendo" := FALSE;
   END_IF;
END_REGION

REGION Network 23
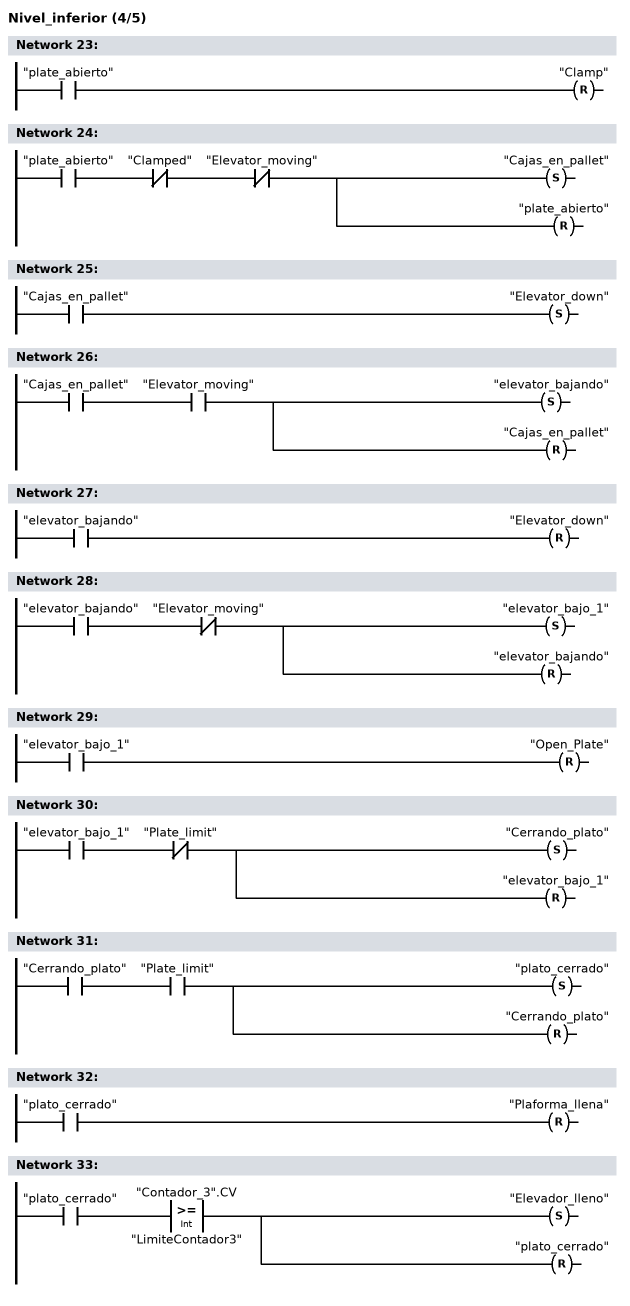
   RUNG wire#powerrail
      Contact( "plate_abierto" )
      R_Coil( "Clamp" )
   END_RUNG
   // the same network as SCL:
   IF "plate_abierto" THEN "Clamp" := FALSE; END_IF;
END_REGION

REGION Network 24
   RUNG wire#powerrail
      Contact( "plate_abierto" )
      I_Contact( "Clamped" )
      I_Contact( "Elevator_moving" )
      wire#w1
      S_Coil( "Cajas_en_pallet" )
   END_RUNG
   RUNG wire#w1
      R_Coil( "plate_abierto" )
   END_RUNG
   // the same network as SCL:
   IF "plate_abierto" AND NOT "Clamped" AND NOT "Elevator_moving" THEN
       "Cajas_en_pallet" := TRUE;
       "plate_abierto" := FALSE;
   END_IF;
END_REGION

REGION Network 25
   RUNG wire#powerrail
      Contact( "Cajas_en_pallet" )
      S_Coil( "Elevator_down" )
   END_RUNG
   // the same network as SCL:
   IF "Cajas_en_pallet" THEN "Elevator_down" := TRUE; END_IF;
END_REGION

REGION Network 26
   RUNG wire#powerrail
      Contact( "Cajas_en_pallet" )
      Contact( "Elevator_moving" )
      wire#w1
      S_Coil( "elevator_bajando" )
   END_RUNG
   RUNG wire#w1
      R_Coil( "Cajas_en_pallet" )
   END_RUNG
   // the same network as SCL:
   IF "Cajas_en_pallet" AND "Elevator_moving" THEN
       "elevator_bajando" := TRUE;
       "Cajas_en_pallet" := FALSE;
   END_IF;
END_REGION

REGION Network 27
   RUNG wire#powerrail
      Contact( "elevator_bajando" )
      R_Coil( "Elevator_down" )
   END_RUNG
   // the same network as SCL:
   IF "elevator_bajando" THEN "Elevator_down" := FALSE; END_IF;
END_REGION

REGION Network 28
   RUNG wire#powerrail
      Contact( "elevator_bajando" )
      I_Contact( "Elevator_moving" )
      wire#w1
      S_Coil( "elevator_bajo_1" )
   END_RUNG
   RUNG wire#w1
      R_Coil( "elevator_bajando" )
   END_RUNG
   // the same network as SCL:
   IF "elevator_bajando" AND NOT "Elevator_moving" THEN
       "elevator_bajo_1" := TRUE;
       "elevator_bajando" := FALSE;
   END_IF;
END_REGION

REGION Network 29
   RUNG wire#powerrail
      Contact( "elevator_bajo_1" )
      R_Coil( "Open_Plate" )
   END_RUNG
   // the same network as SCL:
   IF "elevator_bajo_1" THEN "Open_Plate" := FALSE; END_IF;
END_REGION

REGION Network 30
   RUNG wire#powerrail
      Contact( "elevator_bajo_1" )
      I_Contact( "Plate_limit" )
      wire#w1
      S_Coil( "Cerrando_plato" )
   END_RUNG
   RUNG wire#w1
      R_Coil( "elevator_bajo_1" )
   END_RUNG
   // the same network as SCL:
   IF "elevator_bajo_1" AND NOT "Plate_limit" THEN
       "Cerrando_plato" := TRUE;
       "elevator_bajo_1" := FALSE;
   END_IF;
END_REGION

REGION Network 31
   RUNG wire#powerrail
      Contact( "Cerrando_plato" )
      Contact( "Plate_limit" )
      wire#w1
      S_Coil( "plato_cerrado" )
   END_RUNG
   RUNG wire#w1
      R_Coil( "Cerrando_plato" )
   END_RUNG
   // the same network as SCL:
   IF "Cerrando_plato" AND "Plate_limit" THEN
       "plato_cerrado" := TRUE;
       "Cerrando_plato" := FALSE;
   END_IF;
END_REGION

REGION Network 32
   RUNG wire#powerrail
      Contact( "plato_cerrado" )
      R_Coil( "Plaforma_llena" )
   END_RUNG
   // the same network as SCL:
   IF "plato_cerrado" THEN "Plaforma_llena" := FALSE; END_IF;
END_REGION

REGION Network 33
   RUNG wire#powerrail
      Contact( "plato_cerrado" )
      { S7_Templates := "SrcType := Int" } GE_Contact(in1 := "Contador_3".CV, in2 := "LimiteContador3")
      wire#w1
      S_Coil( "Elevador_lleno" )
   END_RUNG
   RUNG wire#w1
      R_Coil( "plato_cerrado" )
   END_RUNG
   // the same network as SCL:
   IF "plato_cerrado" AND ("Contador_3".CV >= "LimiteContador3") THEN
       "Elevador_lleno" := TRUE;
       "plato_cerrado" := FALSE;
   END_IF;
END_REGION

REGION Network 34
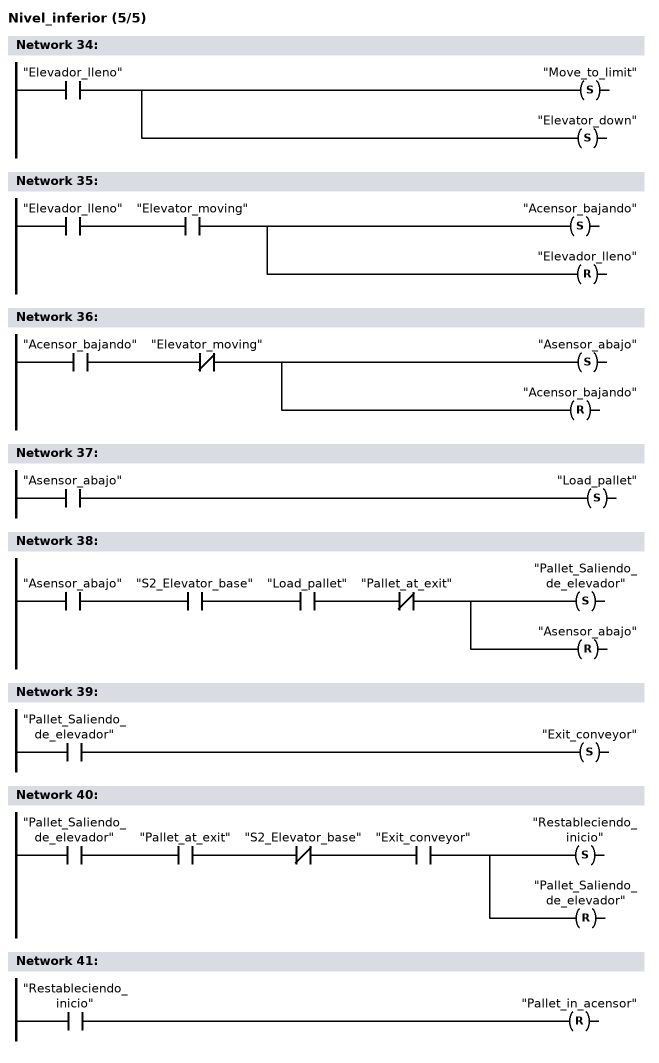
   RUNG wire#powerrail
      Contact( "Elevador_lleno" )
      wire#w1
      S_Coil( "Move_to_limit" )
   END_RUNG
   RUNG wire#w1
      S_Coil( "Elevator_down" )
   END_RUNG
   // the same network as SCL:
   IF "Elevador_lleno" THEN
       "Move_to_limit" := TRUE;
       "Elevator_down" := TRUE;
   END_IF;
END_REGION

REGION Network 35
   RUNG wire#powerrail
      Contact( "Elevador_lleno" )
      Contact( "Elevator_moving" )
      wire#w1
      S_Coil( "Acensor_bajando" )
   END_RUNG
   RUNG wire#w1
      R_Coil( "Elevador_lleno" )
   END_RUNG
   // the same network as SCL:
   IF "Elevador_lleno" AND "Elevator_moving" THEN
       "Acensor_bajando" := TRUE;
       "Elevador_lleno" := FALSE;
   END_IF;
END_REGION

REGION Network 36
   RUNG wire#powerrail
      Contact( "Acensor_bajando" )
      I_Contact( "Elevator_moving" )
      wire#w1
      S_Coil( "Asensor_abajo" )
   END_RUNG
   RUNG wire#w1
      R_Coil( "Acensor_bajando" )
   END_RUNG
   // the same network as SCL:
   IF "Acensor_bajando" AND NOT "Elevator_moving" THEN
       "Asensor_abajo" := TRUE;
       "Acensor_bajando" := FALSE;
   END_IF;
END_REGION

REGION Network 37
   RUNG wire#powerrail
      Contact( "Asensor_abajo" )
      S_Coil( "Load_pallet" )
   END_RUNG
   // the same network as SCL:
   IF "Asensor_abajo" THEN "Load_pallet" := TRUE; END_IF;
END_REGION

REGION Network 38
   RUNG wire#powerrail
      Contact( "Asensor_abajo" )
      Contact( "S2_Elevator_base" )
      Contact( "Load_pallet" )
      I_Contact( "Pallet_at_exit" )
      wire#w1
      S_Coil( "Pallet_Saliendo_de_elevador" )
   END_RUNG
   RUNG wire#w1
      R_Coil( "Asensor_abajo" )
   END_RUNG
   // the same network as SCL:
   IF "Asensor_abajo" AND "S2_Elevator_base" AND "Load_pallet" AND NOT "Pallet_at_exit" THEN
       "Pallet_Saliendo_de_elevador" := TRUE;
       "Asensor_abajo" := FALSE;
   END_IF;
END_REGION

REGION Network 39
   RUNG wire#powerrail
      Contact( "Pallet_Saliendo_de_elevador" )
      S_Coil( "Exit_conveyor" )
   END_RUNG
   // the same network as SCL:
   IF "Pallet_Saliendo_de_elevador" THEN "Exit_conveyor" := TRUE; END_IF;
END_REGION

REGION Network 40
   RUNG wire#powerrail
      Contact( "Pallet_Saliendo_de_elevador" )
      Contact( "Pallet_at_exit" )
      I_Contact( "S2_Elevator_base" )
      Contact( "Exit_conveyor" )
      wire#w1
      S_Coil( "Restableciendo_inicio" )
   END_RUNG
   RUNG wire#w1
      R_Coil( "Pallet_Saliendo_de_elevador" )
   END_RUNG
   // the same network as SCL:
   IF "Pallet_Saliendo_de_elevador" AND "Pallet_at_exit" AND NOT "S2_Elevator_base" AND "Exit_conveyor" THEN
       "Restableciendo_inicio" := TRUE;
       "Pallet_Saliendo_de_elevador" := FALSE;
   END_IF;
END_REGION

REGION Network 41
   RUNG wire#powerrail
      Contact( "Restableciendo_inicio" )
      R_Coil( "Pallet_in_acensor" )
   END_RUNG
   // the same network as SCL:
   IF "Restableciendo_inicio" THEN "Pallet_in_acensor" := FALSE; END_IF;
END_REGION
END_FUNCTION

FUNCTION "Contadores" : Void   // FC3, LAD
{ S7_Optimized_Access := 'TRUE' }
VERSION : 0.1
   VAR_TEMP
      TEMP_salida_conta : Real;
   END_VAR
BEGIN

REGION Network 1
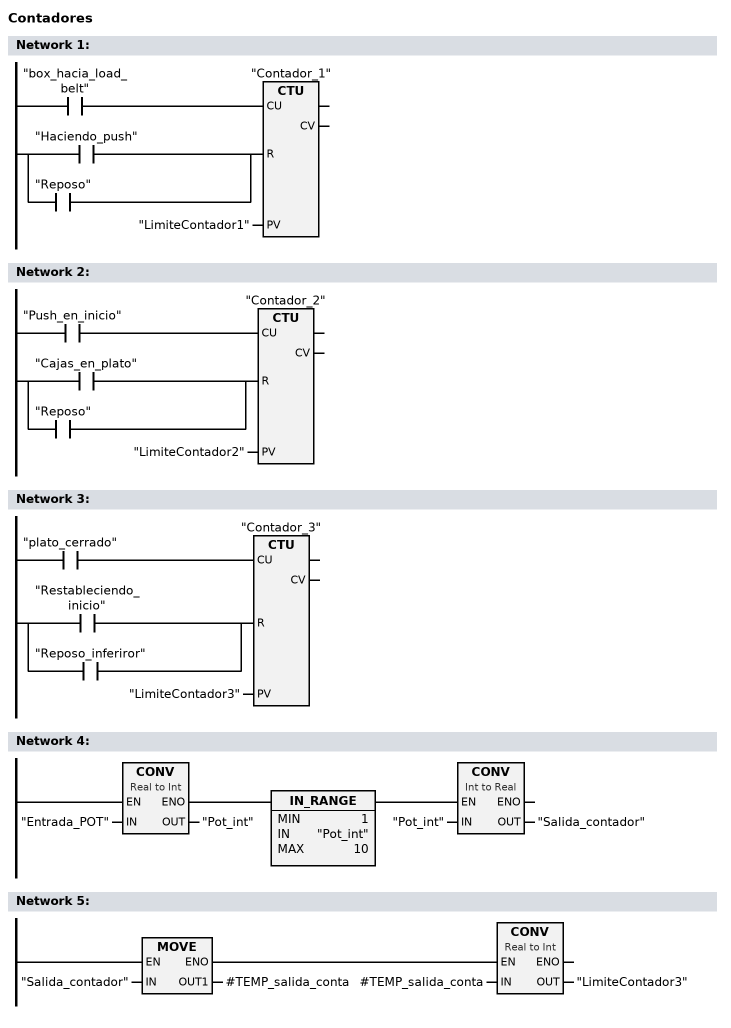
   "Contador_1".CTU(CU := "box_hacia_load_belt", R := "Haciendo_push" OR "Reposo", PV := "LimiteContador1");
END_REGION

REGION Network 2
   "Contador_2".CTU(CU := "Push_en_inicio", R := "Cajas_en_plato" OR "Reposo", PV := "LimiteContador2");
END_REGION

REGION Network 3
   "Contador_3".CTU(CU := "plato_cerrado",
                    R := "Restableciendo_inicio" OR "Reposo_inferiror",
                    PV := "LimiteContador3");
END_REGION

REGION Network 4
   RUNG wire#powerrail
      { S7_Templates := "[SrcType := Real, DestType := Int]" } Convert(in := "Entrada_POT", out => "Pot_int")
      { S7_Templates := "SrcType := Int" } InRange(min := 1, in := "Pot_int", max := 10)
      { S7_Templates := "[SrcType := Int, DestType := Real]" } Convert(in := "Pot_int", out => "Salida_contador")
   END_RUNG
   // the same network as SCL:
   "Pot_int" := REAL_TO_INT("Entrada_POT");
   IF (1 <= "Pot_int") AND ("Pot_int" <= 10) THEN "Salida_contador" := INT_TO_REAL("Pot_int"); END_IF;
END_REGION

REGION Network 5
   RUNG wire#powerrail
      Move(in := "Salida_contador", out1 => #TEMP_salida_conta)
      { S7_Templates := "[SrcType := Real, DestType := Int]" } Convert(in := #TEMP_salida_conta, out => "LimiteContador3")
   END_RUNG
   // the same network as SCL:
   #TEMP_salida_conta := "Salida_contador";
   "LimiteContador3" := REAL_TO_INT(#TEMP_salida_conta);
END_REGION
END_FUNCTION

FUNCTION "Paro emergencia con memoria" : Void   // FC4, LAD
{ S7_Optimized_Access := 'TRUE' }
VERSION : 0.1
   VAR_TEMP
      ParoAux1 : Bool;
      ParoAux2 : Bool;
   END_VAR
   VAR_TEMP   // added for the SCL form of the ladder/FBD networks
      _w1 : Bool;
      _w2 : Bool;
   END_VAR
BEGIN

REGION Network 1
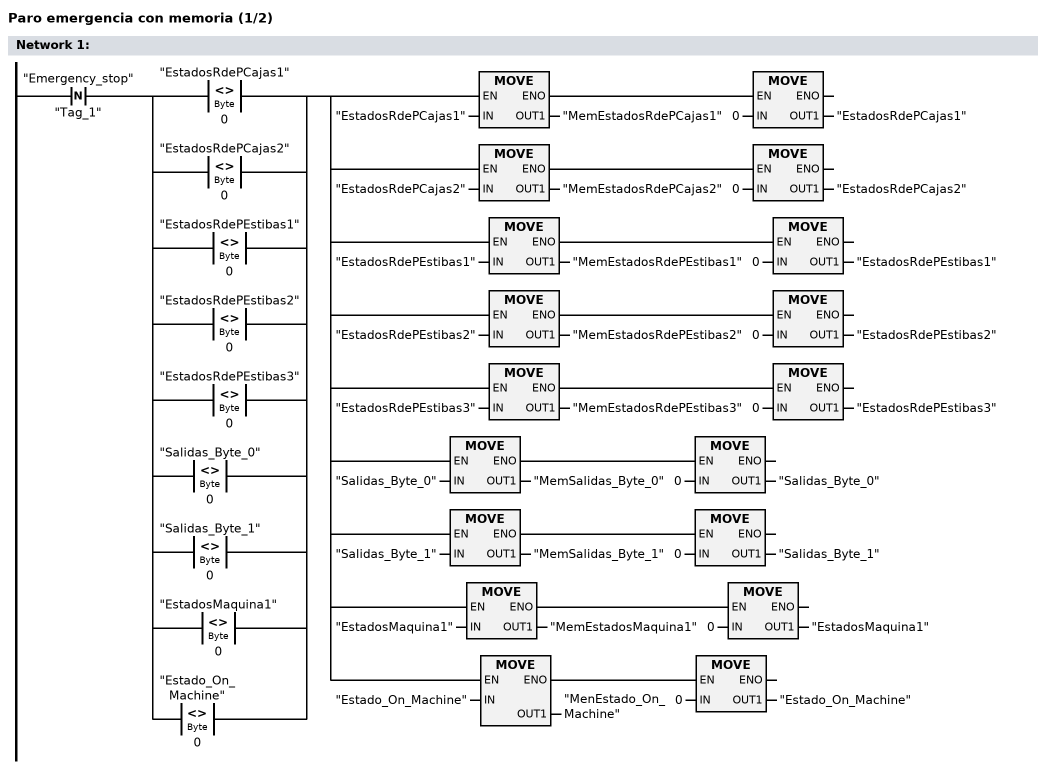
   RUNG wire#powerrail
      N_Contact(operand := "Emergency_stop", bit := "Tag_1")
      wire#w1
      { S7_Templates := "SrcType := Byte" } NE_Contact(in1 := "EstadosRdePCajas1", in2 := 0)
      wire#w2
      Move(in := "EstadosRdePCajas1", out1 => "MemEstadosRdePCajas1")
      Move(in := 0, out1 => "EstadosRdePCajas1")
   END_RUNG
   RUNG wire#w1
      { S7_Templates := "SrcType := Byte" } NE_Contact(in1 := "EstadosRdePCajas2", in2 := 0)
   END_RUNG wire#w2
   RUNG wire#w1
      { S7_Templates := "SrcType := Byte" } NE_Contact(in1 := "EstadosRdePEstibas1", in2 := 0)
   END_RUNG wire#w2
   RUNG wire#w1
      { S7_Templates := "SrcType := Byte" } NE_Contact(in1 := "EstadosRdePEstibas2", in2 := 0)
   END_RUNG wire#w2
   RUNG wire#w1
      { S7_Templates := "SrcType := Byte" } NE_Contact(in1 := "EstadosRdePEstibas3", in2 := 0)
   END_RUNG wire#w2
   RUNG wire#w1
      { S7_Templates := "SrcType := Byte" } NE_Contact(in1 := "Salidas_Byte_0", in2 := 0)
   END_RUNG wire#w2
   RUNG wire#w1
      { S7_Templates := "SrcType := Byte" } NE_Contact(in1 := "Salidas_Byte_1", in2 := 0)
   END_RUNG wire#w2
   RUNG wire#w1
      { S7_Templates := "SrcType := Byte" } NE_Contact(in1 := "EstadosMaquina1", in2 := 0)
   END_RUNG wire#w2
   RUNG wire#w1
      { S7_Templates := "SrcType := Byte" } NE_Contact(in1 := "Estado_On_Machine", in2 := 0)
   END_RUNG wire#w2
   RUNG wire#w2
      Move(in := "EstadosRdePCajas2", out1 => "MemEstadosRdePCajas2")
      Move(in := 0, out1 => "EstadosRdePCajas2")
   END_RUNG
   RUNG wire#w2
      Move(in := "EstadosRdePEstibas1", out1 => "MemEstadosRdePEstibas1")
      Move(in := 0, out1 => "EstadosRdePEstibas1")
   END_RUNG
   RUNG wire#w2
      Move(in := "EstadosRdePEstibas2", out1 => "MemEstadosRdePEstibas2")
      Move(in := 0, out1 => "EstadosRdePEstibas2")
   END_RUNG
   RUNG wire#w2
      Move(in := "EstadosRdePEstibas3", out1 => "MemEstadosRdePEstibas3")
      Move(in := 0, out1 => "EstadosRdePEstibas3")
   END_RUNG
   RUNG wire#w2
      Move(in := "Salidas_Byte_0", out1 => "MemSalidas_Byte_0")
      Move(in := 0, out1 => "Salidas_Byte_0")
   END_RUNG
   RUNG wire#w2
      Move(in := "Salidas_Byte_1", out1 => "MemSalidas_Byte_1")
      Move(in := 0, out1 => "Salidas_Byte_1")
   END_RUNG
   RUNG wire#w2
      Move(in := "EstadosMaquina1", out1 => "MemEstadosMaquina1")
      Move(in := 0, out1 => "EstadosMaquina1")
   END_RUNG
   RUNG wire#w2
      Move(in := "Estado_On_Machine", out1 => "MenEstado_On_Machine")
      Move(in := 0, out1 => "Estado_On_Machine")
   END_RUNG
   // the same network as SCL:
   #_w1 := NOT "Emergency_stop" AND "Tag_1";   // falling edge of "Emergency_stop"
   "Tag_1" := "Emergency_stop";
   IF #_w1 AND (("EstadosRdePCajas1" <> 0) OR ("EstadosRdePCajas2" <> 0) OR ("EstadosRdePEstibas1" <> 0) OR ("EstadosRdePEstibas2" <> 0) OR ("EstadosRdePEstibas3" <> 0) OR ("Salidas_Byte_0" <> 0) OR ("Salidas_Byte_1" <> 0) OR ("EstadosMaquina1" <> 0) OR ("Estado_On_Machine" <> 0)) THEN
       "MemEstadosRdePCajas1" := "EstadosRdePCajas1";
   END_IF;
   #_w2 := #_w1 AND (("EstadosRdePCajas1" <> 0) OR ("EstadosRdePCajas2" <> 0) OR ("EstadosRdePEstibas1" <> 0) OR ("EstadosRdePEstibas2" <> 0) OR ("EstadosRdePEstibas3" <> 0) OR ("Salidas_Byte_0" <> 0) OR ("Salidas_Byte_1" <> 0) OR ("EstadosMaquina1" <> 0) OR ("Estado_On_Machine" <> 0));
   IF #_w2 THEN
       "EstadosRdePCajas1" := 0;
       "MemEstadosRdePCajas2" := "EstadosRdePCajas2";
       "EstadosRdePCajas2" := 0;
       "MemEstadosRdePEstibas1" := "EstadosRdePEstibas1";
       "EstadosRdePEstibas1" := 0;
       "MemEstadosRdePEstibas2" := "EstadosRdePEstibas2";
       "EstadosRdePEstibas2" := 0;
       "MemEstadosRdePEstibas3" := "EstadosRdePEstibas3";
       "EstadosRdePEstibas3" := 0;
       "MemSalidas_Byte_0" := "Salidas_Byte_0";
       "Salidas_Byte_0" := 0;
       "MemSalidas_Byte_1" := "Salidas_Byte_1";
       "Salidas_Byte_1" := 0;
       "MemEstadosMaquina1" := "EstadosMaquina1";
       "EstadosMaquina1" := 0;
       "MenEstado_On_Machine" := "Estado_On_Machine";
       "Estado_On_Machine" := 0;
   END_IF;
END_REGION

REGION Network 2
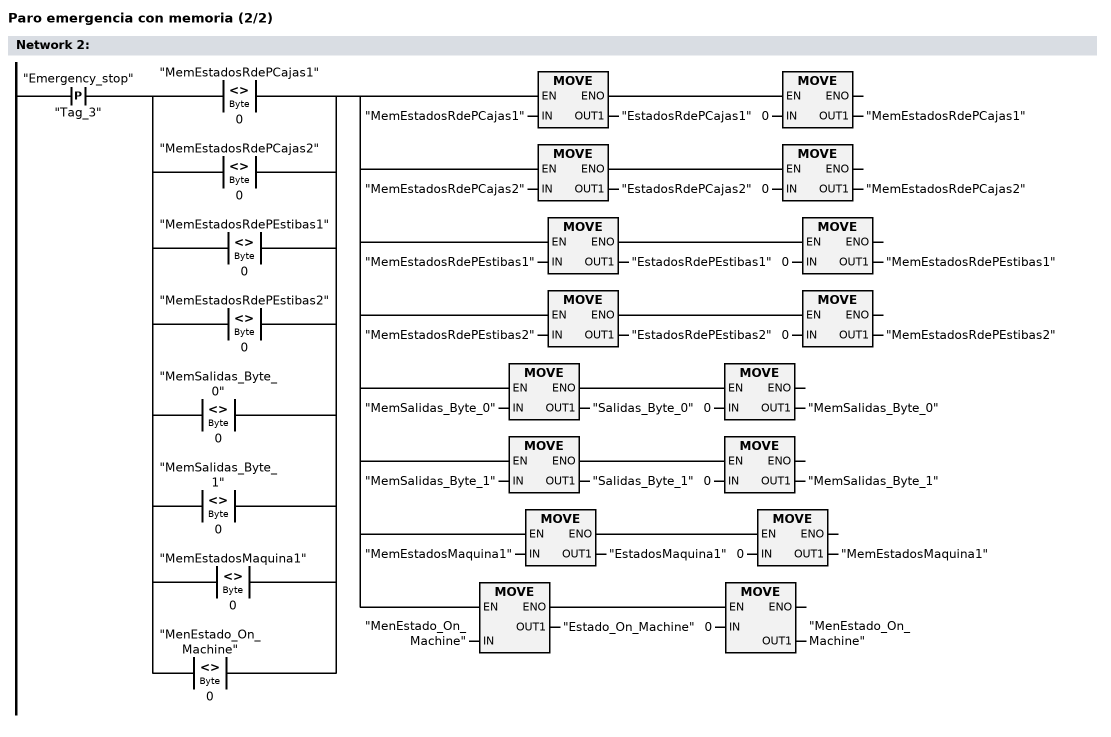
   RUNG wire#powerrail
      P_Contact(operand := "Emergency_stop", bit := "Tag_3")
      wire#w1
      { S7_Templates := "SrcType := Byte" } NE_Contact(in1 := "MemEstadosRdePCajas1", in2 := 0)
      wire#w2
      Move(in := "MemEstadosRdePCajas1", out1 => "EstadosRdePCajas1")
      Move(in := 0, out1 => "MemEstadosRdePCajas1")
   END_RUNG
   RUNG wire#w1
      { S7_Templates := "SrcType := Byte" } NE_Contact(in1 := "MemEstadosRdePCajas2", in2 := 0)
   END_RUNG wire#w2
   RUNG wire#w1
      { S7_Templates := "SrcType := Byte" } NE_Contact(in1 := "MemEstadosRdePEstibas1", in2 := 0)
   END_RUNG wire#w2
   RUNG wire#w1
      { S7_Templates := "SrcType := Byte" } NE_Contact(in1 := "MemEstadosRdePEstibas2", in2 := 0)
   END_RUNG wire#w2
   RUNG wire#w1
      { S7_Templates := "SrcType := Byte" } NE_Contact(in1 := "MemSalidas_Byte_0", in2 := 0)
   END_RUNG wire#w2
   RUNG wire#w1
      { S7_Templates := "SrcType := Byte" } NE_Contact(in1 := "MemSalidas_Byte_1", in2 := 0)
   END_RUNG wire#w2
   RUNG wire#w1
      { S7_Templates := "SrcType := Byte" } NE_Contact(in1 := "MemEstadosMaquina1", in2 := 0)
   END_RUNG wire#w2
   RUNG wire#w1
      { S7_Templates := "SrcType := Byte" } NE_Contact(in1 := "MenEstado_On_Machine", in2 := 0)
   END_RUNG wire#w2
   RUNG wire#w2
      Move(in := "MemEstadosRdePCajas2", out1 => "EstadosRdePCajas2")
      Move(in := 0, out1 => "MemEstadosRdePCajas2")
   END_RUNG
   RUNG wire#w2
      Move(in := "MemEstadosRdePEstibas1", out1 => "EstadosRdePEstibas1")
      Move(in := 0, out1 => "MemEstadosRdePEstibas1")
   END_RUNG
   RUNG wire#w2
      Move(in := "MemEstadosRdePEstibas2", out1 => "EstadosRdePEstibas2")
      Move(in := 0, out1 => "MemEstadosRdePEstibas2")
   END_RUNG
   RUNG wire#w2
      Move(in := "MemSalidas_Byte_0", out1 => "Salidas_Byte_0")
      Move(in := 0, out1 => "MemSalidas_Byte_0")
   END_RUNG
   RUNG wire#w2
      Move(in := "MemSalidas_Byte_1", out1 => "Salidas_Byte_1")
      Move(in := 0, out1 => "MemSalidas_Byte_1")
   END_RUNG
   RUNG wire#w2
      Move(in := "MemEstadosMaquina1", out1 => "EstadosMaquina1")
      Move(in := 0, out1 => "MemEstadosMaquina1")
   END_RUNG
   RUNG wire#w2
      Move(in := "MenEstado_On_Machine", out1 => "Estado_On_Machine")
      Move(in := 0, out1 => "MenEstado_On_Machine")
   END_RUNG
   // the same network as SCL:
   #_w1 := "Emergency_stop" AND NOT "Tag_3";   // rising edge of "Emergency_stop"
   "Tag_3" := "Emergency_stop";
   IF #_w1 AND (("MemEstadosRdePCajas1" <> 0) OR ("MemEstadosRdePCajas2" <> 0) OR ("MemEstadosRdePEstibas1" <> 0) OR ("MemEstadosRdePEstibas2" <> 0) OR ("MemSalidas_Byte_0" <> 0) OR ("MemSalidas_Byte_1" <> 0) OR ("MemEstadosMaquina1" <> 0) OR ("MenEstado_On_Machine" <> 0)) THEN
       "EstadosRdePCajas1" := "MemEstadosRdePCajas1";
   END_IF;
   #_w2 := #_w1 AND (("MemEstadosRdePCajas1" <> 0) OR ("MemEstadosRdePCajas2" <> 0) OR ("MemEstadosRdePEstibas1" <> 0) OR ("MemEstadosRdePEstibas2" <> 0) OR ("MemSalidas_Byte_0" <> 0) OR ("MemSalidas_Byte_1" <> 0) OR ("MemEstadosMaquina1" <> 0) OR ("MenEstado_On_Machine" <> 0));
   IF #_w2 THEN
       "MemEstadosRdePCajas1" := 0;
       "EstadosRdePCajas2" := "MemEstadosRdePCajas2";
       "MemEstadosRdePCajas2" := 0;
       "EstadosRdePEstibas1" := "MemEstadosRdePEstibas1";
       "MemEstadosRdePEstibas1" := 0;
       "EstadosRdePEstibas2" := "MemEstadosRdePEstibas2";
       "MemEstadosRdePEstibas2" := 0;
       "Salidas_Byte_0" := "MemSalidas_Byte_0";
       "MemSalidas_Byte_0" := 0;
       "Salidas_Byte_1" := "MemSalidas_Byte_1";
       "MemSalidas_Byte_1" := 0;
       "EstadosMaquina1" := "MemEstadosMaquina1";
       "MemEstadosMaquina1" := 0;
       "Estado_On_Machine" := "MenEstado_On_Machine";
       "MenEstado_On_Machine" := 0;
   END_IF;
END_REGION
END_FUNCTION

FUNCTION "Manual_Funcion" : Void   // FC5, LAD
{ S7_Optimized_Access := 'TRUE' }
VERSION : 0.1
BEGIN

REGION Network 1
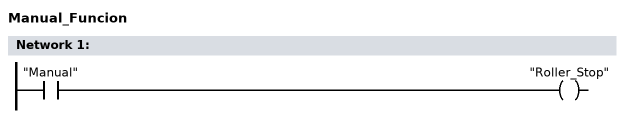
   RUNG wire#powerrail
      Contact( "Manual" )
      Coil( "Roller_Stop" )
   END_RUNG
   // the same network as SCL:
   "Roller_Stop" := "Manual";
END_REGION
END_FUNCTION

FUNCTION "MHJ-PLC-Lab-Function-S71500" : Void   // FC9000, SCL
{ S7_Optimized_Access := 'TRUE' }
VERSION : 0.1
   VAR_TEMP
      Value : Byte;
      ForCounter : Int;
   END_VAR
   VAR CONSTANT
      Value_01_DW : DWord := 16#1223_5486;
      Value_02_DW : DWord := 16#A6C9_D1F5;
   END_VAR
BEGIN

   #Value:=PEEK(area := 16#82,
        dbNumber := 0,
        byteOffset := 511);
   #Value := #Value + 1;

   POKE(area := 16#82,
        dbNumber := 0,
        byteOffset := 511,
        value := #Value);

   POKE(area := 16#82,
        dbNumber := 0,
        byteOffset := 1016,
        value := #Value_01_DW);
   POKE(area := 16#82,
        dbNumber := 0,
        byteOffset := 1020,
        value := #Value_02_DW);

   FOR #ForCounter := 0 TO 63 DO
       #Value:=PEEK(area := 16#1,
            dbNumber := 0,
            byteOffset := #ForCounter);
       POKE(area := 16#81,
            dbNumber := 0,
            byteOffset := #ForCounter,
            value := #Value);
   END_FOR;
   #Value := PEEK(area := 16#1,
                  dbNumber := 0,
                  byteOffset := 512);
   POKE(area := 16#82,
        dbNumber := 0,
        byteOffset := 512,
        value := #Value);
END_FUNCTION

ORGANIZATION_BLOCK "Main"   // OB1, LAD, ProgramCycle
TITLE = "Main Program Sweep (Cycle)"
{ S7_Optimized_Access := 'TRUE' }
VERSION : 0.1
   VAR_INPUT
      Initial_Call : Bool;   // Initial call of this OB
      Remanence : Bool;   // =True, if remanent data are available
   END_VAR
BEGIN

REGION Network 1
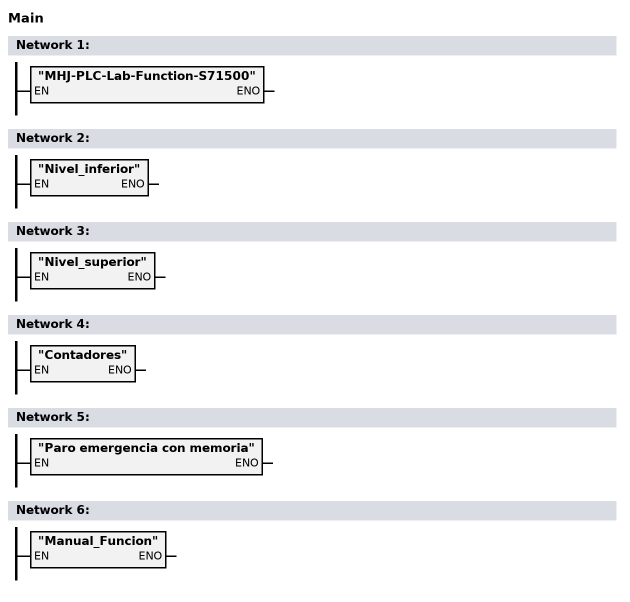
   RUNG wire#powerrail
      "MHJ-PLC-Lab-Function-S71500"()
   END_RUNG
   // the same network as SCL:
   "MHJ-PLC-Lab-Function-S71500"();
END_REGION

REGION Network 2
   RUNG wire#powerrail
      "Nivel_inferior"()
   END_RUNG
   // the same network as SCL:
   "Nivel_inferior"();
END_REGION

REGION Network 3
   RUNG wire#powerrail
      "Nivel_superior"()
   END_RUNG
   // the same network as SCL:
   "Nivel_superior"();
END_REGION

REGION Network 4
   RUNG wire#powerrail
      "Contadores"()
   END_RUNG
   // the same network as SCL:
   "Contadores"();
END_REGION

REGION Network 5
   RUNG wire#powerrail
      "Paro emergencia con memoria"()
   END_RUNG
   // the same network as SCL:
   "Paro emergencia con memoria"();
END_REGION

REGION Network 6
   RUNG wire#powerrail
      "Manual_Funcion"()
   END_RUNG
   // the same network as SCL:
   "Manual_Funcion"();
END_REGION
END_ORGANIZATION_BLOCK

ORGANIZATION_BLOCK "Startup"   // OB100, LAD, Startup
TITLE = "Complete Restart"
{ S7_Optimized_Access := 'TRUE' }
VERSION : 0.1
   VAR_INPUT
      LostRetentive : Bool;   // True if retentive data are lost
      LostRTC : Bool;   // True if date and time are lost
   END_VAR
BEGIN

REGION Network 1
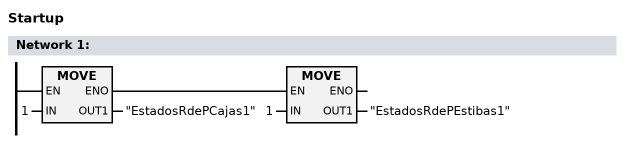
   RUNG wire#powerrail
      Move(in := 1, out1 => "EstadosRdePCajas1")
      Move(in := 1, out1 => "EstadosRdePEstibas1")
   END_RUNG
   // the same network as SCL:
   "EstadosRdePCajas1" := 1;
   "EstadosRdePEstibas1" := 1;
END_REGION
END_ORGANIZATION_BLOCK